Staubli VAL3: gestureWaveout.pgx

program gestureWaveout()
begin
  putln("WaveOut Called")
  movej(wristUp,tClaw,nom_speed)
end
